(* PLC project contactor_2dir_2speed, Dassault Systèmes ControlBuild 2024x *)
(* stored: creationDateTime 2023-10-03T11:13:13-01:00 *)

(* This module simulates control system of motor. This motor has two directions and two speeds. This system is represented by two contactors. *)
FUNCTION_BLOCK equipment_library.contactor_2dir_2speed
  VAR_INPUT
    voltage380 : BOOL := true;
    cmdSupply : BOOL := true;
    sensorSupply : BOOL := true;
  END_VAR
  VAR_INPUT
    forward : BOOL := false;
    backward : BOOL := false;
    highSpeed : BOOL := false;
    lowSpeed : BOOL := false;
  END_VAR
  VAR_OUTPUT
    fwdHsState : BOOL := false;
    fwdLsState : BOOL := false;
    bwdHsState : BOOL := false;
    bwdLsState : BOOL := false;
  END_VAR
  VAR_OUTPUT
    forwardFB : BOOL := false;
    backwardFB : BOOL := false;
    highSpeedFB : BOOL := false;
    lowSpeedFB : BOOL := false;
    thermal : BOOL := false;
  END_VAR
  VAR
    memoFwd : BOOL := false;
    memoBwd : BOOL := false;
    memoLowSpeed : BOOL := false;
    memoHighSpeed : BOOL := false;
  END_VAR
  VAR CONSTANT
    fwdLogic : BOOL := true;
    bwdLogic : BOOL := true;
    highSpeedLogic : BOOL := true;
    lowSpeedLogic : BOOL := true;
    thermalLogic : BOOL := false;
  END_VAR
  VAR
    d_electrical : BOOL := false;
    v_d_electrical : BOOL := false;
    d_Bwd : BOOL := false;
    v_d_Bwd : BOOL := false;
    d_Fwd : BOOL := false;
    v_d_Fwd : BOOL := false;
    d_highSpeed : BOOL := false;
    v_d_highSpeed : BOOL := false;
    d_lowSpeed : BOOL := false;
    v_d_lowSpeed : BOOL := false;
  END_VAR


ACTION C_source_code:
/* ----------------------------------------------------------------	*/
/* Type : Model of Operative Behaviour					*/
/* Category :  Pre-actuators						*/
/* Author : Dassault Systemes						*/
/* Update date : June 2018							*/
/* ----------------------------------------------------------------	*/
/* This module simulates control system of motor. 			*/
/* This motor has two directions and two speeds. 			*/
/* This system is represented by two contactors. 			*/
/* It returns its state and sensors' feed-back.				*/
/* ----------------------------------------------------------------	*/

/* ----------------------------------------------------------------	*/
/* Management of orders from Control Part					*/
/*	if there is no power supply for command 				*/
/*         the contactor doesn't understand the control orders.	*/
/* Contactors can't be actuated at the same time.			*/
/* Security is mchanical.							*/
/* ----------------------------------------------------------------	*/
if (forward && !memoBwd && cmdSupply) memoFwd = 1;
if (!forward || !cmdSupply || d_electrical) memoFwd = 0;
if (!memoFwd && backward && cmdSupply) memoBwd = 1;
if (!backward || !cmdSupply || d_electrical) memoBwd = 0;

if (!memoHighSpeed && lowSpeed && cmdSupply) memoLowSpeed = 1;
if (!lowSpeed || !cmdSupply || d_electrical) memoLowSpeed = 0;
if (highSpeed && !memoLowSpeed && cmdSupply) memoHighSpeed = 1;
if (!highSpeed || !cmdSupply || d_electrical) memoHighSpeed = 0;

/* ----------------------------------------------------------------	*/
/* Calculation of the on-state of contactors				*/
/* ----------------------------------------------------------------	*/
fwdHsState=memoFwd & memoHighSpeed & voltage380;
fwdLsState=memoFwd & memoLowSpeed & ! memoHighSpeed & voltage380;
bwdHsState=memoBwd & memoHighSpeed & voltage380;
bwdLsState=memoBwd & memoLowSpeed & ! memoHighSpeed & voltage380;

/* ----------------------------------------------------------------	*/
/* Management of the thermal feed-back					*/
/* ----------------------------------------------------------------	*/
if (d_electrical) thermal=v_d_electrical;
else
	thermal= ! thermalLogic && sensorSupply;

/* ----------------------------------------------------------------	*/
/* Management of feedback to Control Part					*/
/*     if a fault is required, the contactor feed-back 		*/
/*		 takes a preset state.					*/
/*	if there is no power supply for sensor 				*/
/*         contactor feed-back returns nothing				*/
/*     else contactor feed-back returns the contactor state combined	*/
/*	    with wiring logic.						*/
/* ----------------------------------------------------------------	*/
if (d_Fwd) forwardFB=v_d_Fwd;
else
	forwardFB=(memoFwd ^ ! fwdLogic) && sensorSupply;


if (d_Bwd) backwardFB=v_d_Bwd;
else
	backwardFB=(memoBwd ^ ! bwdLogic) && sensorSupply;


if (d_highSpeed) highSpeedFB=v_d_highSpeed;
else
	highSpeedFB=(memoHighSpeed ^ ! highSpeedLogic) && sensorSupply;


if (d_lowSpeed) lowSpeedFB=v_d_lowSpeed;
else
	lowSpeedFB=(memoLowSpeed ^ ! lowSpeedLogic) && sensorSupply;
END_ACTION
END_FUNCTION_BLOCK
